(* CoDeSys 2.3 export: SYSTEMINFO.exp *)
(* Libraries: STANDARD.LIB 5.6.98 12:03:02, TcBase.lib 14.5.09 12:14:08, TcSystem.lib 21.1.15 10:22:54, TcUtilities.lib 6.1.15 16:45:04 *)

(* POU P_SYSTEMINFO, ST *)
(**************************************************************************************************************)
(*							Beckhoff Automation Poland									*)
(*								P_SYSTEMINFO v2.1									*)
(*									18.09.2015											*)
(* 				v2.1 - dodano zmienne boolowskie okreslajace status 					*)
(* Program odczytuje status systemu, w tym status odczytu zmiennych nieulotnych 		*)
(* Powinien byc wywolany jako pierwszy w pierwszym tasku,							*)
(* a jego satusy powinny byc warunkiem dalszego wykonania programu 					*)
(*________________________________________________________________________*)
PROGRAM P_SYSTEMINFO
VAR
	sStatus				: STRING(8);

	bRetainLOADED		: BOOL;
	bRetainINVALID		: BOOL;
	bRetainREQUESTED	: BOOL;
	bRetainOK			: BOOL;
	bRetainWarning		: BOOL;
	bRetainError		: BOOL;

	bPersistentLOADED	: BOOL;
	bPersistentINVALID	: BOOL;
	bPersistentOK		: BOOL;
	bPersistentWarning	: BOOL;
	bPersistentError		: BOOL;
END_VAR
SYSTEMINFO.runTimeNo;
SYSTEMINFO.projectName;
SYSTEMINFO.numberOfTasks;
SYSTEMINFO.onlineChangeCount;
SYSTEMINFO.systemStateFlags;
SYSTEMINFO.bootDataFlags;
(*Bit number Description
0 RETAIN variables: LOADED (without error) 
1 RETAIN variables: INVALID (the back-up copy was loaded, since no valid data was present) 
2 RETAIN variables: REQUESTED (RETAIN variables should be loaded, a setting in TwinCAT System Control) 
3 reserved 
4 PERSISTENT variables: LOADED (without error) 
5 PERSISTENT variables: INVALID (the back-up copy was loaded, since no valid data was present) 
6 reserved 
7 reserved*)

(* Konwersja na STRING binarnie *)
sStatus := WORD_TO_BINSTR(SYSTEMINFO.bootDataFlags,8);


bRetainLOADED		:= SYSTEMINFO.bootDataFlags.0;
bRetainINVALID		:= SYSTEMINFO.bootDataFlags.1;
bRetainREQUESTED	:= SYSTEMINFO.bootDataFlags.2;

bRetainOK 			:= NOT bRetainREQUESTED OR (bRetainREQUESTED AND NOT bRetainINVALID AND bRetainLOADED); 	(* Status 000 lub 101 *)
bRetainWarning 		:= bRetainREQUESTED AND bRetainINVALID AND bRetainLOADED; 									(* Status 111 *)
bRetainError 		:= bRetainREQUESTED AND bRetainINVALID AND NOT bRetainLOADED; 								(* Status 110 *)

bPersistentLOADED	:= SYSTEMINFO.bootDataFlags.4;
bPersistentINVALID	:= SYSTEMINFO.bootDataFlags.5;

bPersistentOK 		:= NOT bPersistentINVALID AND bPersistentLOADED; 	(* Status 01 *)
bPersistentWarning 	:= bPersistentINVALID AND bPersistentLOADED; 		(* Status 11 *)
bPersistentError 	:= NOT bPersistentOK AND NOT bPersistentWarning; 	(* Status 00 i 10 *)
END_PROGRAM

(* Visualisation SYSTEMINFO
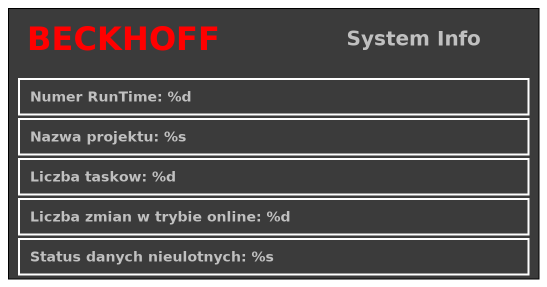
rectangle at (290,0)-(521,61): text "System Info"; dynamic style 16#CCC6BC
rectangle at (10,70)-(521,107): text "Numer RunTime: %d"; shows SystemInfo.runTimeNo
rectangle at (10,110)-(521,147): text "Nazwa projektu: %s"; shows SystemInfo.projectName
rectangle at (10,150)-(521,187): text "Liczba taskow: %d"; shows SystemInfo.numberOfTasks
rectangle at (10,190)-(521,227): text "Liczba zmian w trybie online: %d"; shows SystemInfo.onlineChangeCount
rectangle at (10,230)-(521,267): text "Status danych nieulotnych: %s"; shows P_SYSTEMINFO.sStatus; tooltip Bit number Description 0 RETAIN variables: LOADED (without error) 1 RETAIN variables: INVALID (the back-up copy was loaded, since no valid data was present) 2 RETAIN variables: REQUESTED (RETAIN variables should be loaded, a setting in TwinCAT System Control) 3 reserved 4 PERSISTENT variables: LOADED (without error) 5 PERSISTENT variables: INVALID (the back-up copy was loaded, since no valid data was present) 6 reserved 7 reserved
rectangle at (10,10)-(221,51): text "BECKHOFF"
1 more shapes without text or variables
*)
